{attribute 'GeneratedUsingTerminal: EL7201-0000-0017'}
{attribute addProperty BoxType "EL7201-0000-0017"}
{attribute addProperty Id "FB_PositionAT %I*FB_Position_3FA094ED4DRV_StatuswordAT %I*DRV_Statusword_9B36FDFC2DRV_ControlwordAT %Q*DRV_Controlword_F3F147212DRV_Target_velocityAT %Q*DRV_Target_velocity_08A9583B4WcStateAT %I*WcState_9091E0EB2InfoDataAT %I*InfoData_96C94FAE19"}
{attribute addProperty CRC "3462728655"}
{attribute addProperty Size "33"}
TYPE EL7201_CE650BCF EXTENDS EtcSlaveTerminalBase_947E5A46 :
STRUCT
	{attribute addProperty Name "FB_Position"}
	FB_Position : FB_Position_3FA094ED;
	{attribute addProperty Name "DRV_Statusword"}
	DRV_Statusword : DRV_Statusword_9B36FDFC;
	{attribute addProperty Name "DRV_Controlword"}
	DRV_Controlword : DRV_Controlword_F3F14721;
	{attribute addProperty Name "DRV_Target_velocity"}
	DRV_Target_velocity : DRV_Target_velocity_08A9583B;
	{attribute addProperty Name "WcState"}
	WcState : WcState_9091E0EB;
	{attribute addProperty Name "InfoData"}
	InfoData : InfoData_96C94FAE;
END_STRUCT
END_TYPE

(* stored: Version 1.2.0.0, ProductVersion 3.1.4024.9
   DUT EL7201_CE650BCF: Id {7581ab0c-dba8-4bc2-8c7d-67a8f8d3ac00} *)
